// TIA Portal V20 export
// export: Created 2025-12-01T14:56:09.7167393Z, ExportSetting None, DisplayName Totally Integrated Automation Portal, DisplayVersion V20 Update 3, DisplayName TIA Portal Openness, DisplayVersion V20 Update 3, DisplayName TIA Portal Version Control Interface, DisplayVersion V20 Update 3, DisplayName STEP 7 Professional, DisplayVersion V20 Update 3, DisplayName STEP 7 Safety, DisplayVersion V20 Update 2, DisplayName WinCC Basic/Comfort/Advanced, DisplayVersion V20 Update 3, DisplayName WinCC Professional, DisplayVersion V20 Update 3, DisplayName WinCC Unified, DisplayVersion V20 Update 3
TYPE "LPNDR_typeInterfaceInformation"
   STRUCT
      macAddress : Array[0..5] of Byte;
      nameOfStation : String;
      ipAdress : Array[0..3] of USInt;
      subnetMask : Array[0..3] of USInt;
      gateway : Array[0..3] of USInt;
      mrp { S7_SetPoint := 'True'} : "LPNDR_typeMrpInformation";
   END_STRUCT;
END_TYPE
